# EPICS substitutions: snmpApp/Db/trippLite_pdu_2x.substitutions
file trippLite_pdu_common.db {
{none}
}

file trippLite_pdu_outlet.db {
pattern
{N}
{1}
{2}
}

file misc_common.template {
{none}
}
